# EPICS StreamDevice protocol: Danfysik_HallProbesApp/Db/hallprobe.proto
Terminator = LF;
ReplyTimeout = 2000;
ReadTimeout = 1000;

readField {
    ExtraInput = Ignore;
    in "%*/[^-0-9]*/%f";
}
